TYPE ST_P_ASSY_ELEMENT :
STRUCT
	LeadingSFC:				INT;
	InventoriID:			INT;
END_STRUCT
END_TYPE

(* stored: Version 1.1.0.1, ProductVersion 3.1.4024.10
   DUT ST_P_ASSY_ELEMENT: Id {0d5365ad-8e57-4a56-8dd5-7f50a277ee85} *)
